# EPICS substitutions: IOCs/12id/iocBoot/ioc12ida2/canberra_3.substitutions
file "$(MCA)/mcaApp/Db/simple_mca.db"
{
pattern
{P           M       DTYP           INP              PREC  CHANS}
{12ida2:med:   mca1  "asynMCA"       "@asyn(AIM1/1 0)"  3     2048}
{12ida2:med:   mca2  "asynMCA"       "@asyn(AIM1/2 0)"  3     2048}
{12ida2:med:   mca3  "asynMCA"       "@asyn(AIM2/1 0)"  3     2048}
{12ida2:med:   mca0  "Soft Channel"  ""                 3     2048}
}

#file "$(MCA)/mcaApp/Db/icb_amp.db"
#{
#pattern
#{P			AMP		PORT}
#{12ida2:med:	amp1	icbAmp1}
#}

file "$(MCA)/mcaApp/Db/icb_adc.db"
{
pattern
{P			ADC		PORT}
{12ida2:med:	adc1	"icbAdc1"}
{12ida2:med:	adc2	"icbAdc2"}
{12ida2:med:	adc3	"icbAdc3"}
}

#file "$(MCA)/mcaApp/Db/icb_hvps.db"
#{
#pattern
#{P			HVPS	LIMIT	PORT}
#{12ida2:med:	hvps1	1000	"icbHvps1"}
#}

file "$(MCA)/mcaApp/Db/icb_tca.db"
{
pattern
{P,          TCA,	PORT,		MCA}
{12ida2:med:,  tca1,	"icbTca1",	mca1}
{12ida2:med:,  tca2,	"icbTca2",	mca2}
{12ida2:med:,  tca3,	"icbTca3",	mca3}
}
